RoboDK station: Assistive_UR5e_nou (còpia).rdk

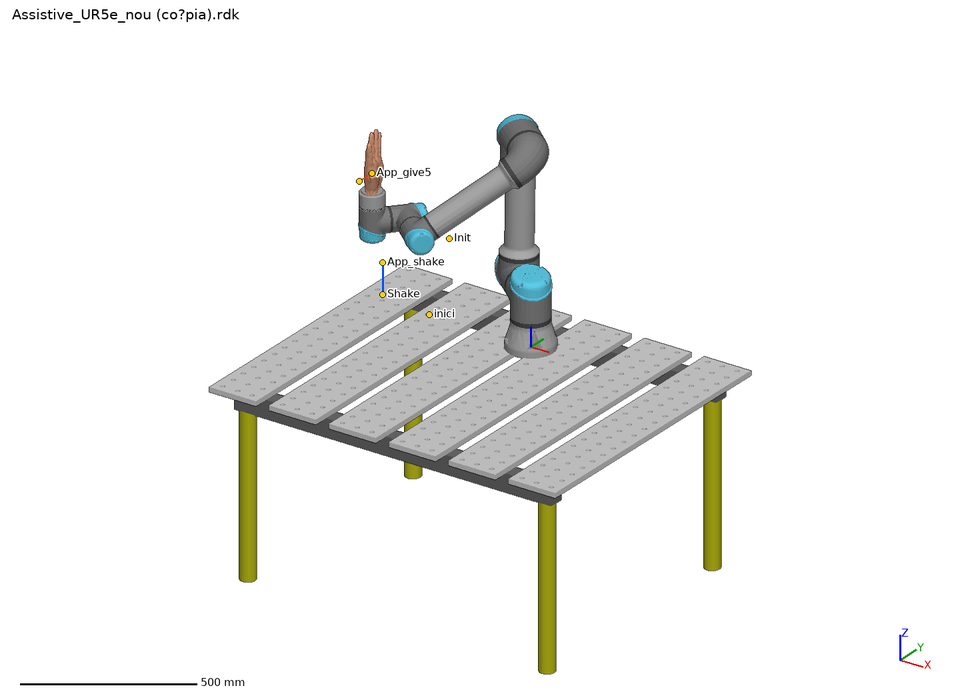
[picture v0: the station drawn from its stored meshes, robots at their saved joint values, targets as dots, program paths as lines]
Station Assistive_UR5e_nou (saved by RoboDK 5.9.2). Poses are relative to the parent item; angles as X-Y-Z fixed-axis rotations.
  - frame UR5e Base at (0, 0, 0) mm
    - robot UR5e: 6 axes, payload 5 kg, reach 850 mm, repeatability 0.03 mm, weight 18.4 kg
        modified DH rows (alpha deg, a mm, theta deg, d mm): 0, 0, 0, 162.5; 90, 0, 180, 0; 0, 425, 0, 0; 0, 392.25, 0, 133.3; -90, 0, 0, 99.7; 90, 0, 180, 99.6
        joint limits [-360, -360, -360, -360, -360, -360] to [360, 360, 360, 360, 360, 360]; home [0, -90, -90, 0, 90, 0]; saved at [-130.679, -89.195, -122.013, 301.208, -90, -119.321]
      - tool Hand, TCP at (0, 0, 50) mm, size 54.8 x 155.9 x 193.5 mm, geometry from Hand.stl
  - frame World at (0, 0, 0) mm
    - object Table at (0, 0, 0) mm, size 1193.8 x 965.2 x 609.6 mm, geometry from welding_table.sld
    - target Init (Cartesian target) at (0, -400, 500) mm, rotated rx 90 ry 0 rz 0 deg; joints [-57.836, -65.392, -107.167, 172.559, -57.836, 0] of UR5e
    - target App_shake (joint target) at (-300, -300, 300) mm, rotated rx 90 ry 0 rz 0 deg; joints [-129.97, -84.968, -123.366, -151.667, -129.97, 0] of UR5e
    - target Shake (joint target) at (-300, -300, 200) mm, rotated rx 90 ry 0 rz 0 deg; joints [-129.97, -95.332, -131.473, -133.195, -129.97, 0] of UR5e
    - target App_give5 (joint target) at (-380.86, -238.62, 533.82) mm, rotated rx 0 ry 0 rz 90 deg; joints [-130.679, -89.195, -122.013, 301.208, -90, 130.679] of UR5e
    - target Give5 (joint target) at (-380.86, -300, 533.82) mm, rotated rx 0 ry 0 rz 90 deg; joints [-125.814, -94.091, -116.939, 301.03, -90, 125.814] of UR5e
    - target inici (Cartesian target) at (0, -500, 300) mm, rotated rx 90 ry 0 rz 0 deg; joints [-292.36, 20.37, -121.299, 100.929, -292.36, 0] of UR5e
    - target ventilar (Cartesian target) at (-380.86, -238.62, 533.82) mm, rotated rx 0 ry 0 rz -160 deg; joints [14.815, 20.403, -90.958, 160.555, -90, 95.185] of UR5e
    - target abaix (Cartesian target) at (-380.86, -238.62, 533.82) mm, rotated rx -4.31 ry -30.91 rz -164.48 deg; joints [-136.691, -101.772, -111.73, 329.548, -107.784, 245.158] of UR5e
  - program Init (3 instructions, listed below)
  - program Hand_shake (5 instructions, listed below)
  - program Give_me_5! (5 instructions, listed below)
  - program MainProgram (4 instructions, listed below)
  - Python program Assistive_hand_SW_nova_funcio (listed below)
  - Python program Assistive_hand_SW_HW_sockets_New (listed below)
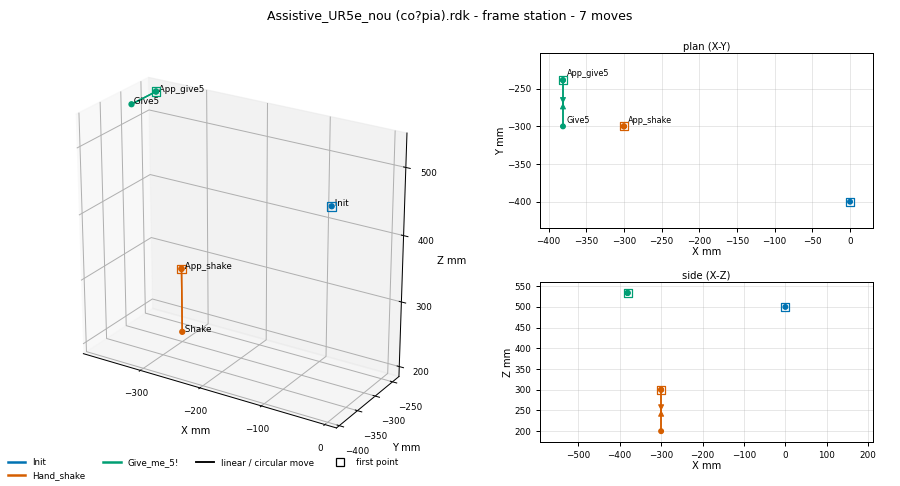
[picture p0: tool path of Assistive_UR5e_nou (còpia).rdk in frame station, 7 of 7 moves have a stored position in this frame; points joined in program order, loops and branches not executed]

--- program Init (robot UR5e) ---
  Est. Ref.: UR5e Base
  Est. herr: Hand
  MoveJ (Init)

--- program Hand_shake (robot UR5e) ---
  Est. Ref.: UR5e Base
  Est. herr: Hand
  MoveL (App_shake)
  MoveL (Shake)
  MoveL (App_shake)

--- program Give_me_5! (robot UR5e) ---
  Est. Ref.: UR5e Base
  Est. herr: Hand
  MoveL (App_give5)
  MoveL (Give5)
  MoveL (App_give5)

--- program MainProgram (robot UR5e) ---
  Llamar Init
  Llamar Hand_shake
  Llamar Give_me_5!
  Llamar Init

--- Python program Assistive_hand_SW_nova_funcio ---
from robodk.robolink import *
from robodk.robomath import *

# Robot setup
RDK = Robolink()
robot = RDK.Item("UR5e")
base = RDK.Item("UR5e Base")
tool = RDK.Item('Hand')
Init_target = RDK.Item('Init')
App_shake_target = RDK.Item('App_shake')
Shake_target = RDK.Item('Shake')
App_give5_target = RDK.Item('App_give5')
Give5_target = RDK.Item('Give5')
#Punts que hem definit nosaltres (nous)
inici_target = RDK.Item('inici')
ventilar_target = RDK.Item('ventilar')
abaix_target = RDK.Item('abaix')

robot.setPoseFrame(base)
robot.setPoseTool(tool)
robot.setSpeed(20)

def Init():
    print("Init")
    robot.MoveL(Init_target, True)
    print("Init_target REACHED")

def Hand_shake():
    print("Hand Shake")
    robot.MoveL(App_shake_target, True)
    robot.MoveL(Shake_target, True)
    robot.MoveL(App_shake_target, True)
    print("Hand Shake FINISHED")

def Give_me_5():
    print("Give me 5!")
    robot.MoveL(App_give5_target, True)
    robot.MoveL(Give5_target, True)
    robot.MoveL(App_give5_target, True)
    print("Give me 5! FINISHED")

def nova_funcio():
    print("Quina calor!")
    robot.MoveL(inici_target, True)
    robot.MoveL(ventilar_target, True)
    robot.MoveL(abaix_target, True)
    robot.MoveL(ventilar_target, True)
    robot.MoveL(abaix_target, True)
    robot.MoveL(ventilar_target, True)
    robot.MoveL(abaix_target, True)
    robot.MoveL(ventilar_target, True)
    print("nova_funcio FINISHED")

# Main function
#def main():
  #  Init()
  #  Hand_shake()
   # Give_me_5()
   # Init()

# Main function
def main():
    nova_funcio()


if __name__ == "__main__":
    main()

--- Python program Assistive_hand_SW_HW_sockets_New ---
import time
from math import radians, degrees, pi
import numpy as np
import socket
#from spatialmath.base import *
from robodk.robolink import *
from robodk.robomath import *

# Robot setup
RDK = Robolink()
robot = RDK.Item("UR5e")
base = RDK.Item("UR5e Base")
tool = RDK.Item('Hand')
Init_target = RDK.Item('Init')
App_shake_target = RDK.Item('App_shake')
Shake_target = RDK.Item('Shake')
App_give5_target = RDK.Item('App_give5')
Give5_target = RDK.Item('Give5')
#Punts que hem definit nosaltres (nous)
inici_target = RDK.Item('inici')
ventilar_target = RDK.Item('ventilar')
abaix_target = RDK.Item('abaix')

# Set robot parameters
robot.setPoseFrame(base)
robot.setPoseTool(tool)
robot.setSpeed(20)

# Robot Constants setup
ROBOT_IP = '192.168.1.5'
ROBOT_PORT = 30002 # Default port for UR robots
accel_mss = 1.2
speed_ms = 0.75
blend_r = 0.0
timej = 6# seconds to finish movej
timel = 4# seconds to finish movel

# Define robot movement commands as URScript strings
set_tcp="set_tcp(p[0.000000, 0.000000, 0.050000, 0.000000, 0.000000, 0.000000])"
movej_init = f"movej([-1.009423, -1.141297, -1.870417, 3.011723, -1.009423, 0.000000],1.20000,0.75000,{timel},0.0000)"
movel_app_shake = f"movel([-2.268404, -1.482966, -2.153143, -2.647089, -2.268404, 0.000000],{accel_mss},{speed_ms},{timel},0.000)"
movel_shake = f"movel([-2.268404, -1.663850, -2.294637, -2.324691, -2.268404, 0.000000],{accel_mss},{speed_ms},{timel/2},0.000)"
movel_app_give5 = f"movel([-2.280779, -1.556743, -2.129529, 5.257071, -1.570796, 2.280779],{accel_mss},{speed_ms},{timel},0.000)"
movel_give5 = f"movel([-2.195869, -1.642206, -2.040971, 5.253965, -1.570796, 2.195869],{accel_mss},{speed_ms},{timel/2},0.000)"
#new robor movement commands
movel_inici = f"movel([    -0.000000,  -500.000000,   300.000000,    90.000000,    -0.000000,    -0.000000 ])"
movel_ventilar = f"movel([  -380.862000,  -238.620000,   533.816000,     0.000000,    -0.000000,  -160.000000 ])"
movel_abaix = f"movel([  -380.862000,  -238.620000,   533.816000,   -45.000000,     0.000000,  -160.000000 ])"

# Initialize UR5e socket communication
def check_robot_port(ROBOT_IP, ROBOT_PORT):
    global robot_socket
    try:
        robot_socket = socket.socket(socket.AF_INET, socket.SOCK_STREAM)
        robot_socket.settimeout(1)  # Tiempo de espera de 1 segundo
        robot_socket.connect((ROBOT_IP, ROBOT_PORT))
        return True
    except (socket.timeout, ConnectionRefusedError):
        return False
# Send commands to the UR5e robot using socket communication
def send_ur_script(command):
    robot_socket.send(("{}\n".format(command)).encode())
def receive_response(t):
    try:
        print("Waiting time: " + str(t))
        time.sleep(t)
    except socket.error as e:
        print(f"Error receiving data from the robot: {e}")
        exit(1) #Non-zero exit status code to indicate the error

def nova_funcio():
    print("Quina calor!")
    robot.MoveL(inici_target, True)
    robot.MoveL(ventilar_target, True)
    robot.MoveL(abaix_target, True)
    robot.MoveL(ventilar_target, True)
    robot.MoveL(abaix_target, True)
    robot.MoveL(ventilar_target, True)
    robot.MoveL(abaix_target, True)
    robot.MoveL(ventilar_target, True)
    print("nova_funcio FINISHED")

    if robot_is_connected:
        print("Ventilar REAL UR5e")
        send_ur_script(set_tcp)
        receive_response(1)
        send_ur_script(movel_inici)
        receive_response(timel)
        send_ur_script(movel_ventilar)
        receive_response(timel)
        send_ur_script(movel_abaix)
        receive_response(timel)
        send_ur_script(movel_ventilar)
        receive_response(timel)
        send_ur_script(movel_abaix)
        receive_response(timel)
        send_ur_script(movel_ventilar)
        receive_response(timel)
        send_ur_script(movel_abaix)
        receive_response(timel)
        send_ur_script(movel_ventilar)
        receive_response(timel)
    else:
        print("UR5e is not connected. Only simulation will take place")


#Main function
def main():
    global robot_is_connected
    robot_is_connected=check_robot_port(ROBOT_IP, ROBOT_PORT)
    nova_funcio()
    if robot_is_connected:
        robot_socket.close()
if __name__ == "__main__":
    main()
